RoboDK station: 新建工作站 (1).rdk

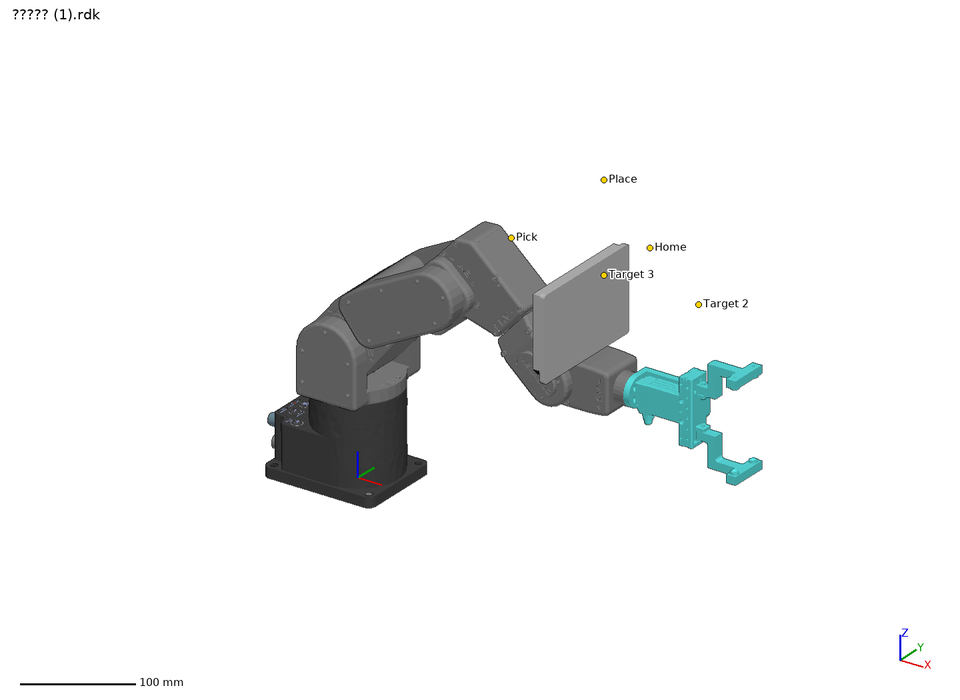
[picture v0: the station drawn from its stored meshes, robots at their saved joint values, targets as dots, program paths as lines]
Station 新建工作站 (1) (saved by RoboDK 6.0.5). Poses are relative to the parent item; angles as X-Y-Z fixed-axis rotations.
  - frame Mecademic Meca500 R4 Base at (0, 0, 0) mm
    - robot Mecademic Meca500 R4: 6 axes
        modified DH rows (alpha deg, a mm, theta deg, d mm): 0, 0, 0, 135; -90, 0, -90, 0; 0, 135, 0, 0; -90, 38, 0, 120; 90, 0, 0, 0; -90, 0, 180, 70
        joint limits [-175, -70, -135, -170, -115, -720] to [175, 90, 70, 170, 115, 720]; home [0, 0, 0, 0, 0, 0]; saved at [0, 52.018, -10.005, 0, -42.013, 90]
      - tool 006., TCP at (0, 0, 119) mm, size 40 x 100.1 x 124.1 mm
    - target Home (joint target) at (309, 0, 308) mm, rotated rx 90 ry 0 rz 90 deg; joints [0, 0, 0, 0, 0, 90] of Mecademic Meca500 R4
    - target Target 2 (Cartesian target) at (290, 100, 208) mm, rotated rx 0 ry 90 rz 0 deg; joints [24.444, 59.102, -43.205, 58.926, -28.89, -55.462] of Mecademic Meca500 R4
    - target Target 3 (Cartesian target) at (190, 100, 208) mm, rotated rx 0 ry 90 rz 0 deg; joints [39.806, 18.561, 24.908, 50.458, -56.115, -34.033] of Mecademic Meca500 R4
    - object 96 at (199, -53, 308) mm, size 14.4 x 127.8 x 85.5 mm, geometry from .STL
    - target Pick (Cartesian target) at (199, -53, 308) mm, rotated rx 90 ry 0 rz 90 deg; joints [-79.315, -26.645, 19.647, 88.683, 79.396, 7.12] of Mecademic Meca500 R4
    - target Place (Cartesian target) at (199, 87, 308) mm, rotated rx 90 ry 0 rz 90 deg; joints [83.443, -13.366, 11.611, 90.202, -83.446, -1.766] of Mecademic Meca500 R4
  - Python program Prog2 (listed below)

--- Python program Prog2 ---
# Type help("robodk.robolink") or help("robodk.robomath") for more information
# Press F5 to run the script
# Documentation: https://robodk.com/doc/en/RoboDK-API.html
# Reference:     https://robodk.com/doc/en/PythonAPI/robodk.html
# Note: It is not required to keep a copy of this file, your Python script is saved with your RDK project

# You can also use the new version of the API:
from robodk import robolink    # RoboDK API
from robodk import robomath    # Robot toolbox
RDK = robolink.Robolink()

# Forward and backwards compatible use of the RoboDK API:
# Remove these 2 lines to follow python programming guidelines
from robodk import *      # RoboDK API
from robolink import *    # Robot toolbox
# Link to RoboDK
# RDK = Robolink()

# Notify user:
print('To edit this program:\nright click on the Python program, then, select "Edit Python script"')

# Program example:
item = RDK.Item('base')
if item.Valid():
    print('Item selected: ' + item.Name())
    print('Item posistion: ' + repr(item.Pose()))

print('Items in the station:')
itemlist = RDK.ItemList()
print(itemlist)

# Provoking an exception will display the console output if you run this script from RoboDK
raise Exception('Program not edited.')
